FUNCTION_BLOCK PUBLIC FB_FAULHABER_SC
VAR_IN_OUT
	Hardware : TYP_FAULHABER_SC_HW;
END_VAR
VAR_INPUT
	AlarmConfig : TYP_ALARM_DEVICE_CONFIG;
	Control : TYP_FAULHABER_SC_CTRL;
END_VAR
VAR_OUTPUT
	Error : BOOL;
END_VAR
VAR
	FaultAlarm : FB_ALARM;
END_VAR

FaultAlarm.Config.Acknowledge := E_ALARM_ACK_TYPE.ACK_AND_RESET;
FaultAlarm.Config.Name := CONCAT(AlarmConfig.Name, '_DRIVE_FAULT');
FaultAlarm(Handler := AlarmConfig.Handler);

IF Hardware.In.Fault THEN
	FaultAlarm.Activate();
END_IF;

Error := Hardware.In.Fault;

IF Control.Run AND Control.Enable THEN
	Hardware.Out.Speed := ABS(Control.Speed);
	Hardware.Out.Direction := Control.Speed >= 0;
ELSE
	Hardware.Out.Speed := 0;
END_IF;

END_FUNCTION_BLOCK

(* stored: Version 1.1.0.1, ProductVersion 3.1.4024.12
   POU FB_FAULHABER_SC: Id {1236047a-c21f-461a-9106-91ab2c1846f9}, SpecialFunc None *)
